% RSLogix 500 project IDENTIFICACION_MOTORCCV_BAK207.RSS, saved by version 7.30.00.17 %
PROJECT "UNTITLED"    % processor: Bul.1763 MicroLogix 1100 Series B %

PROGRAM FILES
  LAD 2 "PRINCIPAL"  5 rungs
  LAD 3 "MODBUS"  5 rungs
  LAD 4 "COMANDOS"  8 rungs
  LAD 5 "HSC_SUB"  6 rungs

DATA FILES
  O0 OUTPUT  4 elements
  I1 INPUT  6 elements
  S2 STATUS  66 elements
  B3 BINARY  1 elements
  T4 TIMER  5 elements
  C5 COUNTER  3 elements
  R6 CONTROL  1 elements
  N7 INTEGER  15 elements
  F8 FLOAT  6 elements
  MG11   5 elements

LADDER 2 "PRINCIPAL"
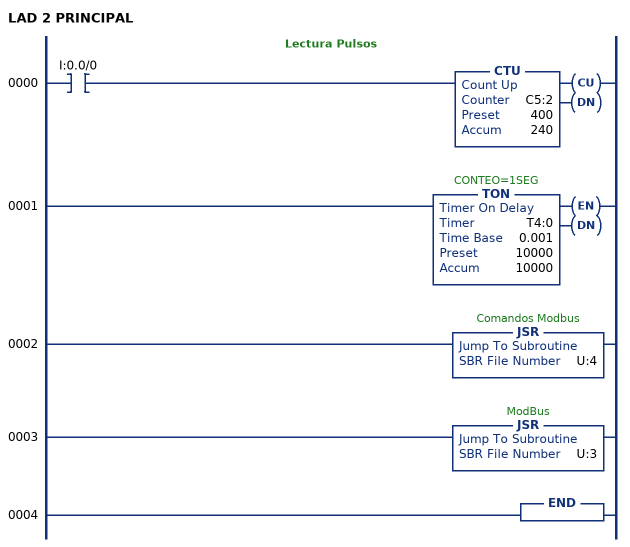
% Rung: 0 %
% TITLE: Lectura Pulsos %
SOR XIC I:0.0/0 CTU C5:2 400 240 EOR
% Rung: 1 %
SOR TON T4:0 0.001 10000 10000 EOR
%   T4:0  "CONTEO=1SEG" %
% Rung: 2 %
SOR JSR U:4 EOR
%   U:4  "Comandos Modbus" %
% Rung: 3 %
SOR JSR U:3 EOR
%   U:3  "ModBus" %
% Rung: 4 %
SOR END EOR

LADDER 3 "MODBUS"
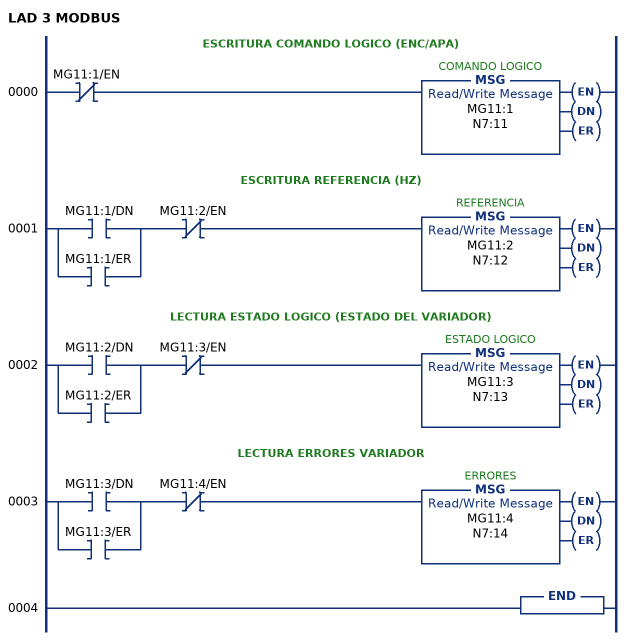
% Rung: 0 %
% TITLE: ESCRITURA COMANDO LOGICO (ENC/APA) %
SOR XIO MG11:1/EN MSG MG11:1 N7:11 EOR
%   MSG set-up: 06 Write Single Register (4xxxxx) | 2 | 1 | 8193 | N7:11 | 0 | 100 | 0 | CLIENT | 0 | 0 | ? %
%   MG11:1  "COMANDO LOGICO" %
%   N7:11  "COMANDO LOGICO" %
% Rung: 1 %
% TITLE: ESCRITURA REFERENCIA (HZ) %
SOR BST XIC MG11:1/DN NXB XIC MG11:1/ER BND XIO MG11:2/EN MSG MG11:2 N7:12 EOR
%   MSG set-up: 06 Write Single Register (4xxxxx) | 2 | 1 | 8194 | N7:12 | 0 | 100 | 0 | CLIENT | 0 | 0 | ? %
%   MG11:2  "REFERENCIA" %
%   N7:12  "REFERENCIA" %
% Rung: 2 %
% TITLE: LECTURA ESTADO LOGICO (ESTADO DEL VARIADOR) %
SOR BST XIC MG11:2/DN NXB XIC MG11:2/ER BND XIO MG11:3/EN MSG MG11:3 N7:13 EOR
%   MSG set-up: 03 Read Holding Registers (4xxxxx) | 2 | 1 | 8449 | N7:13 | 0 | 100 | 0 | CLIENT | 0 | 0 | ? %
%   MG11:3  "ESTADO LOGICO" %
%   N7:13  "ESTADO LOGICO" %
% Rung: 3 %
% TITLE: LECTURA ERRORES VARIADOR %
SOR BST XIC MG11:3/DN NXB XIC MG11:3/ER BND XIO MG11:4/EN MSG MG11:4 N7:14 EOR
%   MSG set-up: 03 Read Holding Registers (4xxxxx) | 2 | 1 | 8450 | N7:14 | 0 | 100 | 0 | CLIENT | 0 | 0 | ? %
%   MG11:4  "ERRORES" %
%   N7:14  "ERRORES" %
% Rung: 4 %
SOR END EOR

LADDER 4 "COMANDOS"
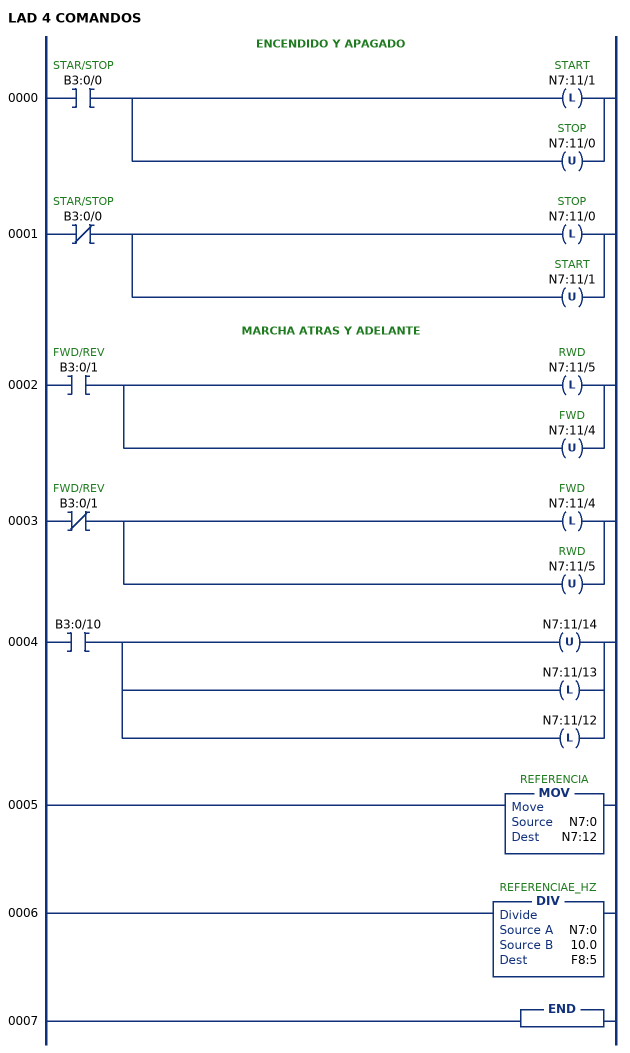
% Rung: 0 %
% TITLE: ENCENDIDO Y APAGADO %
SOR XIC B3:0/0 BST OTL N7:11/1 NXB OTU N7:11/0 BND EOR
%   B3:0/0  "STAR/STOP" %
%   N7:11/1  "START" %
%   N7:11/0  "STOP" %
% Rung: 1 %
SOR XIO B3:0/0 BST OTL N7:11/0 NXB OTU N7:11/1 BND EOR
%   B3:0/0  "STAR/STOP" %
%   N7:11/0  "STOP" %
%   N7:11/1  "START" %
% Rung: 2 %
% TITLE: MARCHA ATRAS Y ADELANTE %
SOR XIC B3:0/1 BST OTL N7:11/5 NXB OTU N7:11/4 BND EOR
%   B3:0/1  "FWD/REV" %
%   N7:11/5  "RWD" %
%   N7:11/4  "FWD" %
% Rung: 3 %
SOR XIO B3:0/1 BST OTL N7:11/4 NXB OTU N7:11/5 BND EOR
%   B3:0/1  "FWD/REV" %
%   N7:11/4  "FWD" %
%   N7:11/5  "RWD" %
% Rung: 4 %
SOR XIC B3:0/10 BST OTU N7:11/14 NXB OTL N7:11/13 NXB OTL N7:11/12 BND EOR
% Rung: 5 %
SOR MOV N7:0 N7:12 EOR
%   N7:0  "SP-FRECUENCIA" %
%   N7:12  "REFERENCIA" %
% Rung: 6 %
SOR DIV N7:0 10.0 F8:5 EOR
%   N7:0  "SP-FRECUENCIA" %
%   F8:5  REFERENCIAE_HZ %
% Rung: 7 %
SOR END EOR

LADDER 5 "HSC_SUB"
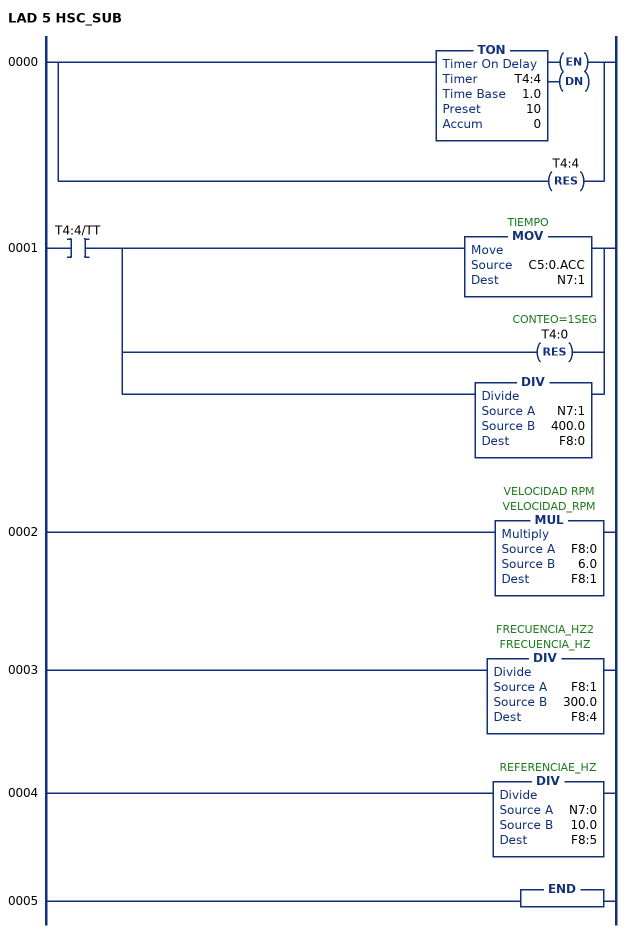
% Rung: 0 %
SOR BST TON T4:4 1.0 10 0 NXB RES T4:4 BND EOR
% Rung: 1 %
SOR XIC T4:4/TT BST MOV C5:0.ACC N7:1 NXB RES T4:0 NXB DIV N7:1 400.0 F8:0 BND EOR
%   N7:1  "TIEMPO" %
%   T4:0  "CONTEO=1SEG" %
% Rung: 2 %
SOR MUL F8:0 6.0 F8:1 EOR
%   F8:1  VELOCIDAD_RPM  "VELOCIDAD RPM" %
% Rung: 3 %
SOR DIV F8:1 300.0 F8:4 EOR
%   F8:1  VELOCIDAD_RPM  "VELOCIDAD RPM" %
%   F8:4  FRECUENCIA_HZ  "FRECUENCIA_HZ2" %
% Rung: 4 %
SOR DIV N7:0 10.0 F8:5 EOR
%   N7:0  "SP-FRECUENCIA" %
%   F8:5  REFERENCIAE_HZ %
% Rung: 5 %
SOR END EOR

OTHER DOCUMENTED ADDRESSES
  F8:3  "FRECUENCIA_HZ1"
  N7:2  REFERENCIA_HZ
  PFILE:5  "HSC"
  U:5  "HSC"

COMMENTS NOT ATTACHED TO A CURRENT RUNG
  MG11:4: FALLAS
  MG11:3: FRECUENCIA
  MG11:2: DATOS DE ESTADO LOGICO
  MG11:1: REFERENCIA
  MG11:0: ESCRITURA COMANDO LOGICO (ENC/APA)
  N12:0/2: JOG
  N12:0/5: FWD

DATA TABLE (non-zero values as saved)
DATA B3
% B3:0 % 0X0412
DATA T4
% .PRE .ACC %
% T4:0 % 10000 10000
% T4:4 % 10 0
DATA C5
% .PRE .ACC %
% C5:2 % 400 240
DATA N7
% N7:0 % 450 403 0 0 0 0 0 0 0 0
% N7:10 % 0 12321 450 1537 0
DATA F8
% F8:0 % 2.475248 540.9357 54093.57 0 19.43016
% F8:5 % 45
